{attribute 'hide_all_locals'}
FUNCTION F_Compare : BOOL
VAR_INPUT
	fValueA 		: REAL;
	fValueB 		: REAL;
	fTolerance 		: REAL := 1E-6;	
END_VAR

VAR
	fDifference 	: REAL;
END_VAR

fDifference := ABS(fValueB - fValueA);
fTolerance := LIMIT(1E-6, ABS(fTolerance), 1E+6);
F_Compare := fTolerance > fDifference;

END_FUNCTION

(* stored: Version 1.1.0.1, ProductVersion 3.1.4024.12
   POU F_Compare: Id {806b9cee-6c90-0d48-3903-6abca9e7f319}, SpecialFunc None *)
